FUNCTION F_ULINT_RTN : ULINT
VAR_INPUT
	stArg : ST_Arg;
END_VAR
VAR
	sysVar_Info : __SYSTEM.VAR_INFO;
END_VAR

sysVar_Info := __VARINFO(F_ULINT_RTN);
IF stArg.TypeClass = sysVar_Info.TypeClass THEN 
	F_ULINT_RTN := TO_ULINT(stArg.sValue);
	END_IF

END_FUNCTION

(* stored: Version 1.1.0.1, ProductVersion 3.1.4024.4
   POU F_ULINT_RTN: Id {7ba2dd9c-871d-4cfd-8f6a-1108b3c419cc}, SpecialFunc None *)
